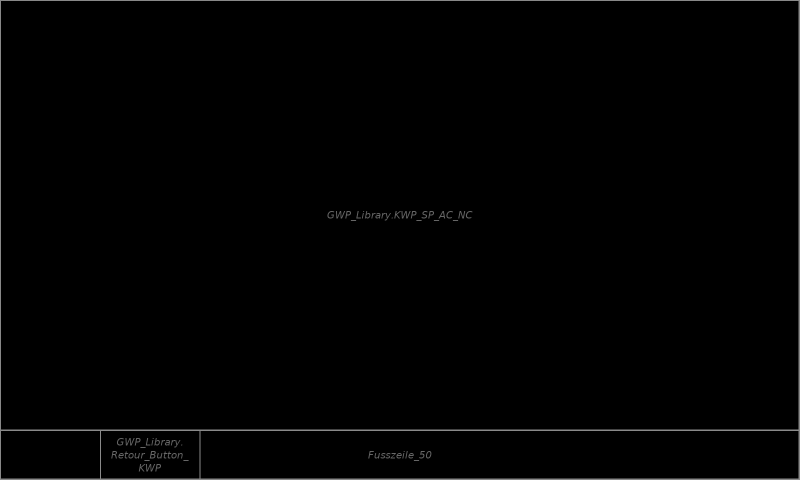
VISUALIZATION KWP_SP_AC_NC  // 800x480
    Frame (0,0 800x430)
        shows GWP_Library.KWP_SP_AC_NC(FB_KWP_SP_AC_NC := Main.KWP_SP_AC_NC_0, FB_Kreis_3KO := Main.Kreis_3KO_0, FB_VD := Main.VD_0)
    Group (0,430 800x50)
        Frame (0,0 800x50)
            shows Fusszeile_50()
        Frame (100,0 100x50)
            shows GWP_Library.Retour_Button_KWP()
END_VISUALIZATION

(* stored: Version 1.1.0.1, ProductVersion 3.1.4022.6
   Visu KWP_SP_AC_NC: Id {2be4b5e1-6981-473f-bd06-3a53ba3eb378} *)
